Fanuc KAREL source: kt00416.compact.KL

PROGRAM KT00416
%STACKSIZE=65535
%PRIORITY=65535
%NOLOCKGROUP
VAR
H1 : ARRAY[2] OF SHORT
R2 : REAL
OUT : BOOLEAN
BEGIN
H1[1]=2
R2=3.0
OUT=((H1[1]) > R2)
END KT00416
